# EPICS autosave request: iocs/zwoIOC/iocBoot/iocZWODriver/auto_settings.req
file "ZWODriver_settings.req",    P=$(P),  R=cam1:
file "NDStdArrays_settings.req",  P=$(P),  R=image1:
